(* PLC project Generated.project, CODESYS CODESYS V3.5 SP19 Patch 1 *)
(* stored: creationDateTime 2026-11-18T13:59:46.966479, modificationDateTime 2026-11-18T13:59:46.966479 *)

(* ======================================================================= 💾 ST_Encoder_Calib — Calibration & référence codeur (1 par treuil, RETAIN) ─────────────────────────────────────────────────────────────── 🎯 Rôle : Structure de calibration RETAIN par treuil (M1_EncoderCalib / M2_EncoderCalib) 💾 Données : Références brutes, état homed et contrôle de cohérence redémarrage 📄 Doc métier : DOC/AF/AF_Partie-09_Fonction_Encoder_v2.4.md ======================================================================= *)
TYPE ST_Encoder_Calib : STRUCT
  HomingRefRaw : UDINT;  (* === DONNEES DE REFERENCE BRUTE (RETAIN) === Valeur brute figee au dernier homing reussi *)
  LastKnownRawPos : UDINT;  (* Dernier point brut valide connu (continu) *)
  RestartCoherenceTolerancePts : UDINT := 1000;  (* === CONFIGURATION & REGLAGES TOLERANCE === Tolerance redemarrage (pts, ~12% de 8192) *)
  Homed : BOOL;  (* === ETATS DE CALIBRATION & SECURITE === TRUE des qu'un referencement a reussi *)
  HomingSuspect : BOOL;  (* TRUE si incoherence detectee au redemarrage *)
  HomingProvisional : BOOL;  (* TRUE si zero provisoire 0m HX1 (avant HX4 8.5m) *)
END_STRUCT;
END_TYPE

(* ======================================================================= 🧩 ST_Fault — Brique socle défaut (2 vues : live + latchée) ─────────────────────────────────────────────────────────────── 🎯 Rôle : porter l'état défaut d'un composant, applicable dans TOUS les cas (acquittable ou non), sans brique warning séparée. • Vue LIVE (Error / ErrorId) : suit la cause, retombe seule à 0. • Vue LATCHÉE (Latched / LatchedId): mémorisée au défaut, reste jusqu'au front Reset. Le choix acquittable / non-acquittable se fait PAR CAUSE (ST_FaultCause.Latching), jamais par bloc. 🔒 Sécurité : interlock TOUJOURS sur la cause brute (Error / ErrorId), jamais sur l'acquittement. Reset TOUJOURS effectif, jamais conditionné (std §9). 🧬 Composition : brique de base réutilisable — sortie de FB, struct métier, GVL. Texte IHM NON stocké ici : dérivé côté IHM depuis LatchedId / ErrorId. 📄 Doc : DOC/STDS/CODE_QUALITY_STANDARDS.md §2quinquies / §9 ======================================================================= *)
TYPE ST_Fault : STRUCT
  Error : BOOL;  (* <-- [DIAG] vue LIVE : au moins une cause présente maintenant *)
  ErrorId : WORD;  (* <-- [DIAG] bitfield des causes présentes maintenant (0 si aucune) *)
  Latched : BOOL;  (* <-- [DIAG] vue LATCHÉE : défaut non acquitté, reste jusqu'au front Reset *)
  LatchedId : WORD;  (* <-- [DIAG] ErrorId figé à l'apparition du défaut, effacé au Reset *)
END_STRUCT;
END_TYPE

(* ======================================================================= 🧩 ST_FaultCause — Cause élémentaire alimentant ST_Fault (socle FB_FaultCore) ─────────────────────────────────────────────────────────────── 🎯 Rôle : une cause exprimée EN CLAIR (BOOL + libellé), sans bitfield ni masque. Le FB métier remplit une liste (ARRAY[0..15] OF ST_FaultCause) ; le socle FB_FaultCore en déduit ST_Fault (vue live + vue latchée). 🔒 Sécurité : interlock TOUJOURS sur Active (cause brute), jamais sur le latch. Latching = TRUE → la cause ARME la vue latchée (défaut à acquitter). Latching = FALSE → la cause n'alimente que la vue live (retombe seule). Fail-safe : une cause laissée à Latching=FALSE reste visible en live — pour la rendre acquittable, il faut le déclarer explicitement. 📄 Doc : DOC/STDS/CODE_QUALITY_STANDARDS.md §2quinquies / §9 ======================================================================= *)
TYPE ST_FaultCause : STRUCT
  Active : BOOL;  (* 1 = cause présente maintenant (interlock sur cette valeur) *)
  Latching : BOOL;  (* 1 = cause à acquitter (arme Latched) ; 0 = live seulement *)
  Texte : STRING;  (* libellé prêt IHM (non stocké dans ST_Fault, dérivé côté IHM) *)
END_STRUCT;
END_TYPE

(* ======================================================================= 🧩 ST_Lifecycle — Brique socle cycle d'exécution ─────────────────────────────────────────────────────────────── 🎯 Rôle : porter l'avancement d'une action à cycle (organe, séquenceur). Optionnelle : un FB purement synchrone (conditionneur, filtre, joystick) ne la porte pas. 🧬 Composition : brique de base réutilisable, composée avec ST_Fault. 📄 Doc : DOC/STDS/CODE_QUALITY_STANDARDS.md §2quinquies ======================================================================= *)
TYPE ST_Lifecycle : STRUCT
  Busy : BOOL;  (* <-- [STAT] 1 = action en cours *)
  Done : BOOL;  (* <-- [STAT] 1 = action terminée avec succès *)
END_STRUCT;
END_TYPE

(* ======================================================================= ⚙️ ST_fbEncoder_Cfg — Réglages technologiques publics de FB_Encoder ─────────────────────────────────────────────────────────────────────── 🎯 Rôle : porter le mode de confirmation preset commun aux codeurs. 🔒 Ownership : GVL_IHM.Commun.EncoderCfg ↔ GVL_PERSISTENT._EncoderCfgPersist. 📄 Doc : DOC/AF/AF_Partie-09_Fonction_Encoder_v2.4.md ======================================================================= *)
TYPE ST_fbEncoder_Cfg : STRUCT
  PresetConfirmMode : E_PresetConfirmMode := E_PresetConfirmMode.READBACK_ONLY;  (* Mode de confirmation preset, défaut relecture *)
  Initialized : BOOL := FALSE;  (* 🚦 TRUE après restauration du pont persistant *)
END_STRUCT;
END_TYPE

(* values of E_PresetConfirmMode: READBACK_ONLY: Confirmation par relecture de position; READBACK_AND_STATUSBIT: Relecture et bit d'état matériel; STATUSBIT_ONLY: Bit d'état matériel uniquement *)

{attribute 'qualified_only'}
{attribute 'strict'}
TYPE E_PresetConfirmMode : (READBACK_ONLY := 0, READBACK_AND_STATUSBIT := 1, STATUSBIT_ONLY := 2);
END_TYPE

(* ======================================================================= ⚙️ FB_Encoder_Homing — Référencement codeur nominal ou unitaire ─────────────────────────────────────────────────────────────── 🎯 Rôle : Séquence de référencement nominal (capteur haut) ou unitaire (MAINT_N2) 🔒 Polarité : Homed=TRUE dès qu'un référencement valide est enregistré 🔌 Architecture : Expose ST_Encoder_Calib en VAR_IN_OUT 📄 Doc métier : DOC/AF/AF_Partie-09_Fonction_Encoder_v2.4.md ======================================================================= === DECLARATION (à coller dans la partie déclaration du POU FB_Encoder_Homing) === *)
FUNCTION_BLOCK FB_Encoder_Homing
  VAR_INPUT
    Enable : BOOL;  (* === COMMANDES & AUTORISATIONS === --> [CMD] Autorisation generale FB (TRUE=Autorise) *)
    Reset : BOOL;  (* --> [CMD] Acquittement defaut (front montant) *)
    Home : BOOL;  (* --> [CMD] Demande de referencement (front) *)
    HomingPermit : BOOL;  (* --> [CMD] Autorisation de homer (calculee par le caller) *)
    BtnConfirmCoherence : BOOL;  (* --> [CMD] Levee de doute d'incoherence au boot (front) *)
    InvalidateDatum : BOOL := FALSE;  (* --> [CMD] Invalidation explicite du datum (abandon avant calibration finale) *)
    ProvisionalHoming : BOOL := FALSE;  (* --> [CMD] TRUE = preset provisoire (ex. 0m HX1), FALSE = definitif *)
    CfgHomingTargetM : REAL;  (* === CIBLES & CONFIGURATION HOMING === --> [CFG] Cible libre homing unitaire (m) *)
    UseDynamicTarget : BOOL := FALSE;  (* --> [CFG] Activation cible dynamique *)
    DynamicHomingTargetM : REAL := 0;  (* --> [CFG] Cible dynamique de referencement (m) *)
    CfgTopSensorPosM : REAL := 8.5;  (* --> [CFG] Cible homing nominal capteur haut (m) *)
    TopPositionSensor : BOOL;  (* === RETOURS HW & CAPTEURS === --> [HW] Capteur physique position haute unique *)
    RawPos : UDINT;  (* === MESURES & RETOURS FB CODEUR ABSOLU === --> [HW] Position brute codeur (sortie FB_Encoder_Abs) *)
    EncoderAvailable : BOOL;  (* --> [HW] Codeur absolu disponible et valide *)
    PresetStatusBit : BOOL;  (* --> [HW] Bit d'etat preset optionnel, FALSE si non cable *)
    Cfg : ST_fbEncoder_Cfg;  (* === REGLAGES TRANSACTION PRESET === --> [CFG] Mode de confirmation preset *)
    PointsPerRev : UDINT := 8192;  (* === CARACTERISTIQUES MECANIQUES & BUS === --> [CFG] Resolution codeur (pts/tour) *)
    MultiTurnRevsMax : UDINT := 4096;  (* --> [CFG] Capacite multitour max codeur (tours) *)
    CableM_PerRev : REAL := 2;  (* --> [CFG] Perimetre tambour / developpement cable (m/tour) *)
    BypassGlobal : BOOL := FALSE;  (* === TESTS & BYPASS === --> [TST] Neutralisation securites pour mise en service *)
  END_VAR
  VAR_OUTPUT
    Ready : BOOL;  (* === ETATS IEC & SYNOPTIQUE === <-- [STAT] FB pret a fonctionner *)
    Fault : ST_Fault;  (* 🧩 Statut transverse (forme cible ST_Fault) *)
    Lifecycle : ST_Lifecycle;  (* 🧩 Cycle de vie (forme cible ST_Lifecycle) *)
    PresetRequest : BOOL;  (* === COMMANDES VERS FB_ENCODER_ABS === <-- [ACT] Pulse demande d'ecriture preset SDO *)
    PresetValue : UDINT;  (* <-- [ACT] Valeur de cible brute pour preset SDO *)
    Homed : BOOL;  (* === RESULTATS & MEMOIRE CALIBRATION === <-- [STAT] Codeur pagine et referencie *)
    HomingSuspect : BOOL;  (* <-- [DIAG] Incoherence redemarrage a lever *)
    HomingProvisional : BOOL;  (* <-- [STAT] TRUE si datum provisoire RETAIN actif (HX1 0m) *)
    HomingRefRaw : UDINT;  (* <-- [DIAG] Offset de reference brut calcule *)
    PresetConfirmationFailed : BOOL;  (* <-- [DIAG] Latch derniere verification preset echouee *)
  END_VAR
  VAR_IN_OUT
    Calib : ST_Encoder_Calib;  (* === STRUCTURE DE CALIBRATION PERSISTANTE === <-> [BUS] Structure de calibration RETAIN *)
  END_VAR
  VAR
    ResetEdge : R_TRIG;  (* === DETECTEURS DE FRONT === . [LOC] Detecteur front montant Reset *)
    HomeEdge : R_TRIG;  (* . [LOC] Detecteur front montant Home *)
    ConfirmCoherenceEdge : R_TRIG;  (* . [LOC] Detecteur front montant BtnConfirmCoherence *)
    TopSensorEdge : R_TRIG;  (* . [LOC] Detecteur front montant TopPositionSensor *)
    DynamicTargetEdge : R_TRIG;  (* . [LOC] Detecteur front montant UseDynamicTarget *)
    InitDone : BOOL;  (* === ETATS & DRAPEAUX INTERNES === . [LOC] Controle incoherence boot effectue *)
    HomingModeOk : BOOL;  (* . [LOC] Mode de fonctionnement valide pour homing *)
    NominalHomingTrigger : BOOL;  (* . [LOC] Condition de declenchement homing nominal *)
    UnitaryHomingTrigger : BOOL;  (* . [LOC] Condition de declenchement homing unitaire *)
    DynamicHomingTrigger : BOOL;  (* . [LOC] Condition de declenchement homing dynamique *)
    HomingTrigger : BOOL;  (* . [LOC] Synthese declenchement homing *)
    PresetVerificationActive : BOOL;  (* . [LOC] Verification preset en attente *)
    PendingProvisional : BOOL;  (* . [LOC] Capture mode provisoire pendant verification preset *)
    PresetConfirmed : BOOL;  (* . [LOC] Resultat du mode de confirmation selectionne *)
    HomingModeError : BOOL;  (* === DRAPEAUX DEFAUTS INTERNES === . [LOC] Latch erreur mode *)
    TargetOutOfRangeError : BOOL;  (* . [LOC] Latch cible hors limites *)
    PresetFailError : BOOL;  (* . [LOC] Latch échec preset *)
    BootIncoherentError : BOOL;  (* . [LOC] Latch incohérence boot *)
    TargetPoints : DINT;  (* === VARIABLES DE CALCUL === . [LOC] Ecart cible converti en points *)
    TargetPositionM : REAL;  (* . [LOC] Cible retenue en metres *)
    RawDiffRestart : DINT;  (* . [LOC] Ecart brut de position au redemarrage *)
    PendingHomingRefRaw : UDINT;  (* . [LOC] Reference candidate, non publiee avant succes *)
    CandidateRawDiff : DINT;  (* . [LOC] Ecart brut de la mesure candidate *)
    CandidateCablePosM : REAL;  (* . [LOC] Position candidate calculee avant commit *)
    ReadbackOk : BOOL;  (* . [LOC] Mesure candidate dans la tolerance *)
    StatusBitOk : BOOL;  (* . [LOC] Etat du bit optionnel de confirmation *)
    PresetVerifyTimer : TON;  (* . [LOC] Temporisation historique de verification 500ms *)
    instFault : FB_FaultCore;  (* === SOCLE DEFAUT (FB_FaultCore) === * [INST] Socle défaut transverse *)
    instCauses : ARRAY[0..15] OF ST_FaultCause;  (* . [LOC] Table des causes nommées *)
    CST_HomingVerifyToleranceM : REAL := 0.01;  (* === TOLERANCE & TEMPORISATION TRANSACTION === Tolerance mesure cible (m) *)
    CST_PresetVerifyTime : TIME := TIME#50MS;  (* Latence historique avant relecture *)
  END_VAR

            

// === IMPLEMENTATION (à coller dans le corps ST du POU FB_Encoder_Homing) ===

{region "§1 Causes & Socle Défaut (évalué en continu)"}
// 🔑 1. FRONTS
ResetEdge(CLK := Reset);
HomeEdge(CLK := Home);
ConfirmCoherenceEdge(CLK := BtnConfirmCoherence);

// Effacement des latches d'erreur sur Reset conscient
IF ResetEdge.Q THEN
    PresetConfirmationFailed := FALSE;
    HomingModeError := FALSE;
    TargetOutOfRangeError := FALSE;
    PresetFailError := FALSE;
END_IF;

// Levée de doute incohérence boot (BtnConfirmCoherence)
IF ConfirmCoherenceEdge.Q THEN
    Calib.HomingSuspect := FALSE;
    BootIncoherentError := FALSE;
END_IF;

// Configuration des causes nommées
instCauses[0].Active   := HomingModeError;
instCauses[0].Latching := TRUE;
instCauses[0].Texte    := 'Homing non autorise dans ce mode';

instCauses[1].Active   := TargetOutOfRangeError;
instCauses[1].Latching := TRUE;
instCauses[1].Texte    := 'Cible de homing hors plage';

instCauses[2].Active   := PresetFailError;
instCauses[2].Latching := TRUE;
instCauses[2].Texte    := 'Echec confirmation transaction preset';

instCauses[3].Active   := BootIncoherentError;
instCauses[3].Latching := TRUE;
instCauses[3].Texte    := 'Incoherence position codeur au demarrage';

// Appel du socle de défaut
instFault(Enable := Enable, Reset := Reset, Causes := instCauses);
Fault := instFault.Fault;
{endregion}

{region "§2 Gate neutralisation"}
// 🛑 2. GATE — neutralisation ; on continue toutefois d'exposer le dernier état RETAIN connu
// (FB_Encoder_Scale a besoin de HomingRefRaw même si ce FB est désactivé)
IF NOT Enable THEN
    PresetRequest := FALSE;
    PresetValue := 0;
    Ready := FALSE;
    Lifecycle.Busy := FALSE;
    Lifecycle.Done := FALSE;
    InitDone := FALSE;   // Force un nouveau contrôle à la prochaine activation
    PresetVerificationActive := FALSE;
    PresetVerifyTimer(IN := FALSE, PT := CST_PresetVerifyTime);
    Homed := Calib.Homed;
    HomingSuspect := Calib.HomingSuspect;
    HomingProvisional := Calib.HomingProvisional;
    HomingRefRaw := Calib.HomingRefRaw;
    // PresetConfirmationFailed est un diagnostic latch : il est gelé hors Enable
    RETURN;
END_IF;

Ready := Enable AND NOT Fault.Latched;
{endregion}

IF InvalidateDatum THEN
    Calib.Homed              := FALSE;
    Calib.HomingSuspect      := FALSE;
    Calib.HomingProvisional  := FALSE;
    PendingProvisional       := FALSE;
    Lifecycle.Done           := FALSE;
    PresetVerificationActive := FALSE;
    PresetVerifyTimer(IN := FALSE, PT := CST_PresetVerifyTime);
END_IF;

{region "§3 Cohérence au redémarrage"}
// 🔍 3. COHÉRENCE AU REDÉMARRAGE — une fois par session Enable, dès que le codeur répond
IF NOT InitDone THEN
    IF EncoderAvailable THEN
        RawDiffRestart := UDINT_TO_DINT(RawPos) - UDINT_TO_DINT(Calib.LastKnownRawPos);
        IF Calib.Homed AND (ABS(RawDiffRestart) > UDINT_TO_DINT(Calib.RestartCoherenceTolerancePts)) THEN
            Calib.HomingSuspect := TRUE;
            BootIncoherentError := TRUE;
        END_IF;
        InitDone := TRUE;
    END_IF;
END_IF;
{endregion}

{region "§4 Demande et déclenchement homing"}
// ⚙️ 4. DEMANDE & DÉCLENCHEMENT HOMING
PresetRequest := FALSE;
PresetValue := 0;
TopSensorEdge(CLK := TopPositionSensor);
DynamicTargetEdge(CLK := UseDynamicTarget);

HomingModeOk := HomingPermit;

IF HomeEdge.Q AND NOT HomingModeOk THEN
    HomingModeError := TRUE;
END_IF;

NominalHomingTrigger := HomingModeOk AND NOT UseDynamicTarget
                         AND ((Home AND TopSensorEdge.Q) OR (HomeEdge.Q AND TopPositionSensor));

UnitaryHomingTrigger := HomingModeOk AND NOT UseDynamicTarget AND HomeEdge.Q;

DynamicHomingTrigger := HomingModeOk AND (DynamicTargetEdge.Q OR (UseDynamicTarget AND HomeEdge.Q));

HomingTrigger := (NominalHomingTrigger OR UnitaryHomingTrigger OR DynamicHomingTrigger)
                 AND NOT PresetVerificationActive;

IF HomingTrigger THEN
    IF UseDynamicTarget THEN
        TargetPositionM := DynamicHomingTargetM;
    ELSIF NominalHomingTrigger THEN
        TargetPositionM := CfgTopSensorPosM;
    ELSE
        TargetPositionM := CfgHomingTargetM;
    END_IF;

    // Bornage obligatoire avant écriture (CODE_QUALITY_STANDARDS §6) [-99;+99] m
    IF (TargetPositionM < -99.0) OR (TargetPositionM > 99.0) THEN
        TargetOutOfRangeError := TRUE;
    ELSE
        TargetPoints := REAL_TO_DINT(TargetPositionM * UDINT_TO_REAL(PointsPerRev) / CableM_PerRev);
        PendingHomingRefRaw := DINT_TO_UDINT(UDINT_TO_DINT(RawPos) - TargetPoints);
        PresetValue := RawPos;
        PresetRequest := TRUE;
        PresetVerificationActive := TRUE;
        PendingProvisional := ProvisionalHoming;
        Lifecycle.Done := FALSE;
    END_IF;
END_IF;
{endregion}

{region "§5 Suivi de transaction preset"}
// ⏳ 5. SUIVI DE LA TRANSACTION PRESET
PresetVerifyTimer(IN := PresetVerificationActive, PT := CST_PresetVerifyTime);
IF PresetVerificationActive AND PresetVerifyTimer.Q THEN
    CandidateRawDiff := UDINT_TO_DINT(RawPos) - UDINT_TO_DINT(PendingHomingRefRaw);
    IF PointsPerRev <> 0 THEN
        CandidateCablePosM := DINT_TO_REAL(CandidateRawDiff) * CableM_PerRev / UDINT_TO_REAL(PointsPerRev);
    ELSE
        CandidateCablePosM := 0.0;
    END_IF;
    ReadbackOk := ABS(CandidateCablePosM - TargetPositionM) <= CST_HomingVerifyToleranceM;
    StatusBitOk := PresetStatusBit;

    CASE Cfg.PresetConfirmMode OF
        E_PresetConfirmMode.READBACK_ONLY:
            PresetConfirmed := ReadbackOk;
        E_PresetConfirmMode.READBACK_AND_STATUSBIT:
            PresetConfirmed := ReadbackOk AND StatusBitOk;
        E_PresetConfirmMode.STATUSBIT_ONLY:
            PresetConfirmed := StatusBitOk;
        ELSE
            PresetConfirmed := FALSE;
    END_CASE;

    IF PresetConfirmed THEN
        Calib.HomingRefRaw := PendingHomingRefRaw;
        Calib.Homed := TRUE;
        Calib.HomingSuspect := FALSE;
        Calib.HomingProvisional := PendingProvisional;
        Calib.LastKnownRawPos := RawPos;
        PresetConfirmationFailed := FALSE;
        PresetFailError := FALSE;
        Lifecycle.Done := TRUE;
    ELSE
        Calib.HomingSuspect := TRUE;
        Calib.HomingProvisional := FALSE;
        PresetConfirmationFailed := TRUE;
        PresetFailError := TRUE;
        Lifecycle.Done := FALSE;
    END_IF;

    PendingProvisional := FALSE;
    PresetVerificationActive := FALSE;
    PresetVerifyTimer(IN := FALSE, PT := CST_PresetVerifyTime);
END_IF;
{endregion}

{region "§6 Sorties état & calibration"}
// 📤 6. SORTIES ÉTAT & CALIBRATION
IF EncoderAvailable AND NOT PresetVerificationActive THEN
    Calib.LastKnownRawPos := RawPos;
END_IF;

Lifecycle.Busy := PresetVerificationActive;
Homed := Calib.Homed AND NOT Calib.HomingSuspect;
HomingSuspect := Calib.HomingSuspect;
HomingProvisional := Calib.HomingProvisional;
HomingRefRaw := Calib.HomingRefRaw;
{endregion}

          
END_FUNCTION_BLOCK

(* ======================================================================= 🧩 FB_FaultCore — Socle de remplissage de ST_Fault (vue live + vue latchée) ─────────────────────────────────────────────────────────────── 🎯 Rôle : à partir d'une LISTE de causes en clair (ARRAY[0..15] OF ST_FaultCause), produire la brique ST_Fault : • Error / ErrorId : vue LIVE, suit les causes Active, retombe seule. • Latched / LatchedId: vue LATCHÉE, chaque bit figé à l'apparition d'une cause `Active AND Latching`, conservé jusqu'au front Reset. 🔒 Sécurité : - interlock TOUJOURS sur `Causes[i].Active` (cause brute), jamais sur le latch. - Reset TOUJOURS effectif, jamais conditionné (std §9) — agit même Enable=FALSE. - Latching=FALSE → cause visible en LIVE seulement (fail-safe : reste visible). - un défaut laté non acquitté reste publié même FB désactivé (pas d'effacement silencieux sur bascule Enable OFF→ON sans Reset). - une cause à acquitter réapparue re-arme son bit (ré-alarme). 🧬 Un seul socle, réutilisé par tout FB `standard` qui expose un ST_Fault. Pas de State, pas de Warning, pas de texte — hors périmètre de ce socle. 📄 Doc : DOC/STDS/CODE_QUALITY_STANDARDS.md §2quinquies / §9 ======================================================================= *)
FUNCTION_BLOCK FB_FaultCore
  VAR_INPUT
    Enable : BOOL;  (* --> [CMD] Autorisation générale du FB porteur *)
    Reset : BOOL;  (* --> [CMD] Front d'acquittement (jamais conditionné, §9) *)
    Causes : ARRAY[0..15] OF ST_FaultCause;  (* --> [CMD] Liste des causes en clair (Active / Latching / Texte) *)
  END_VAR
  VAR_OUTPUT
    Ready : BOOL;  (* <-- [STAT] FB porteur autorisé (= Enable) *)
    Fault : ST_Fault;  (* <-- [DIAG] Brique défaut (mappée 1:1 sur la sortie du FB porteur) *)
  END_VAR
  VAR
    ResetEdge : R_TRIG;  (* . [LOC] Front montant Reset *)
    Latch : ARRAY[0..15] OF BOOL;  (* . [LOC] Bit laté par cause, jusqu'au Reset *)
    i : INT;  (* . [LOC] Index de parcours de la liste *)
  END_VAR

            

{region "§1 Reset (front, toujours effectif)"}
// Front Reset : efface tous les latches. Jamais conditionné, agit même Enable=FALSE (§9).
Ready := Enable;
ResetEdge(CLK := Reset);
IF ResetEdge.Q THEN
    FOR i := 0 TO 15 DO Latch[i] := FALSE; END_FOR;
END_IF;
{endregion}

{region "§2 Vue LIVE — Error / ErrorId"}
// Bitfield des causes présentes MAINTENANT. Retombe seule à 0 quand les causes disparaissent.
// Non évaluée si Enable=FALSE (pas de lecture de cause hors autorisation).
Fault.ErrorId := 0;
IF Enable THEN
    FOR i := 0 TO 15 DO
        IF Causes[i].Active THEN
            Fault.ErrorId := Fault.ErrorId OR SHL(WORD#1, INT_TO_DWORD(i));
        END_IF;
    END_FOR;
END_IF;
Fault.Error := (Fault.ErrorId <> 0);
{endregion}

{region "§3 Armement des latches (causes à acquitter)"}
// Une cause Active ET Latching arme son bit ; le bit reste jusqu'au front Reset (§1),
// même si la cause disparaît. Réapparition => ré-armement (ré-alarme).
IF Enable THEN
    FOR i := 0 TO 15 DO
        IF Causes[i].Active AND Causes[i].Latching THEN
            Latch[i] := TRUE;
        END_IF;
    END_FOR;
END_IF;
{endregion}

{region "§4 Vue LATCHÉE — Latched / LatchedId"}
// Toujours publiée, y compris Enable=FALSE : un défaut non acquitté reste visible.
Fault.LatchedId := 0;
FOR i := 0 TO 15 DO
    IF Latch[i] THEN
        Fault.LatchedId := Fault.LatchedId OR SHL(WORD#1, INT_TO_DWORD(i));
    END_IF;
END_FOR;
Fault.Latched := (Fault.LatchedId <> 0);
{endregion}

          
END_FUNCTION_BLOCK
